// TIA Portal project "CAMASIR_MAKINASI" (V15.1)

(* hardware
DEVICE "S7300/ET200M station_1"  S7-300 station
   slot 0: "Rail_0"  Rail  6ES7 390-1***0-0AA0
   slot 2: "PLC_1"  CPU 314C-2 PN/DP  6ES7 314-6EH04-0AB0  V3.3
      slot 2: "PROFINET interface_1"  PN-IO
         slot 1: "Port_1"  Port
         slot 2: "Port_2"  Port
      slot 5: "DI 24/DO 16_1"  DI24/DO16
      slot 6: "AI 5/AO 2_1"  AI5/AO2
      slot 7: "Count_1"  Counter
      slot 8: "Positioning_1"  Positioning
*)

// ===== PLC "PLC_1"  CPU 314C-2 PN/DP =====

VAR_GLOBAL   // PLC tag table "Default tag table"
   "START" AT %I0.0 : Bool;
   "LAMBA" AT %Q0.0 : Bool;
   "STOP" AT %I0.1 : Bool;
   "V1" AT %Q0.1 : Bool;
   "L" AT %I0.2 : Bool;
   "H" AT %I0.3 : Bool;
   "Tag_1" AT %M0.0 : Bool;
   "Tag_2" AT %M1.0 : Bool;
   "Tag_3" AT %M0.1 : Bool;
   "Tag_4" AT %M1.1 : Bool;
   "Tag_5" AT %I0.7 : Bool;
   "Tag_6" AT %MW1 : Int;
   "V3" AT %Q0.2 : Bool;
   "L1" AT %I0.4 : Bool;
   "H1" AT %I0.5 : Bool;
   "Tag_7" AT %M0.2 : Bool;
   "Tag_8" AT %M1.2 : Bool;
   "Tag_9" AT %I0.6 : Bool;
   "Tag_10" AT %M0.3 : Bool;
   "Tag_11" AT %M1.3 : Bool;
   "M1" AT %Q0.3 : Bool;
   "L2" AT %I1.0 : Bool;
   "H2" AT %I1.1 : Bool;
   "Tag_12" AT %M0.4 : Bool;
   "Tag_13" AT %M1.4 : Bool;
   "Tag_14" AT %M0.5 : Bool;
   "Tag_15" AT %M1.5 : Bool;
   "V2" AT %Q0.6 : Bool;
   "L3" AT %I1.2 : Bool;
   "H3" AT %I1.3 : Bool;
   "Tag_16" AT %M0.6 : Bool;
   "Tag_17" AT %M1.6 : Bool;
   "Tag_18" AT %MW2 : Int;
   "Tag_19" AT %M2.2 : Bool;
   "Tag_20" AT %M2.3 : Bool;
   "Tag_21" AT %MW3 : Int;
   "Tag_22" AT %M1.7 : Bool;
   "Tag_23" AT %M2.0 : Bool;
   "Tag_24" AT %M2.1 : Bool;
END_VAR

ORGANIZATION_BLOCK "Main"   // OB1, LAD
TITLE = "Main Program Sweep (Cycle)"
{ S7_Optimized_Access := 'FALSE' }
VERSION : 0.1
   VAR_TEMP
      OB1_EV_CLASS : Byte;   // Bits 0-3 = 1 (Coming event), Bits 4-7 = 1 (Event class 1)
      OB1_SCAN_1 : Byte;   // 1 (Cold restart scan 1 of OB 1), 3 (Scan 2-n of OB 1)
      OB1_PRIORITY : Byte;   // Priority of OB Execution
      OB1_OB_NUMBR : Byte;   // 1 (Organization block 1, OB1)
      OB1_RESERVED_1 : Byte;   // Reserved for system
      OB1_RESERVED_2 : Byte;   // Reserved for system
      OB1_PREV_CYCLE : Int;   // Cycle time of previous OB1 scan (milliseconds)
      OB1_MIN_CYCLE : Int;   // Minimum cycle time of OB1 (milliseconds)
      OB1_MAX_CYCLE : Int;   // Maximum cycle time of OB1 (milliseconds)
      OB1_DATE_TIME : Date_And_Time;   // Date and time OB1 started
   END_VAR
   VAR_TEMP   // added for the SCL form of the ladder/FBD networks
      _w1 : Bool;
   END_VAR
BEGIN

REGION Network 1
   // START LAMA
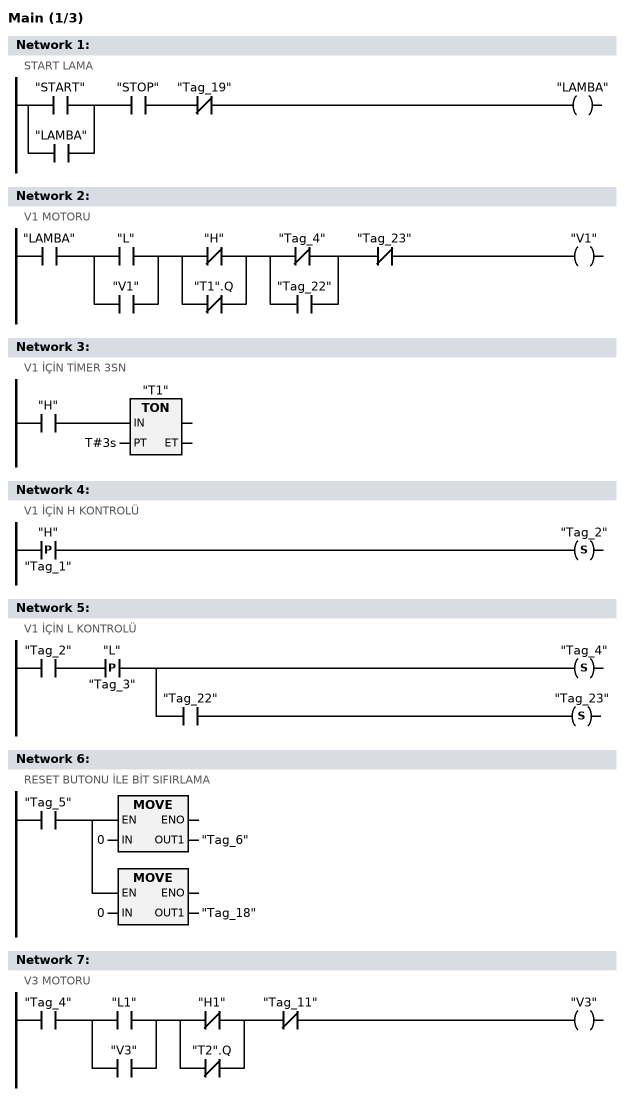
   RUNG wire#powerrail
      Contact( "START" )
      wire#w1
      Contact( "STOP" )
      I_Contact( "Tag_19" )
      Coil( "LAMBA" )
   END_RUNG
   RUNG wire#powerrail
      Contact( "LAMBA" )
   END_RUNG wire#w1
   // the same network as SCL:
   "LAMBA" := ("START" OR "LAMBA") AND "STOP" AND NOT "Tag_19";
END_REGION

REGION Network 2
   // V1 MOTORU
   RUNG wire#powerrail
      Contact( "LAMBA" )
      wire#w1
      Contact( "L" )
      wire#w2
      I_Contact( "H" )
      wire#w3
      I_Contact( "Tag_4" )
      wire#w4
      I_Contact( "Tag_23" )
      Coil( "V1" )
   END_RUNG
   RUNG wire#w1
      Contact( "V1" )
   END_RUNG wire#w2
   RUNG wire#w2
      I_Contact( "T1".Q )
   END_RUNG wire#w3
   RUNG wire#w3
      Contact( "Tag_22" )
   END_RUNG wire#w4
   // the same network as SCL:
   "V1" := "LAMBA" AND ("L" OR "V1") AND (NOT "H" OR NOT "T1".Q) AND (NOT "Tag_4" OR "Tag_22") AND NOT "Tag_23";
END_REGION

REGION Network 3
   // V1 İÇİN TİMER 3SN
   "T1".TON(IN := "H", PT := T#3s);
END_REGION

REGION Network 4
   // V1 İÇİN H KONTROLÜ
   RUNG wire#powerrail
      P_Contact(operand := "H", bit := "Tag_1")
      S_Coil( "Tag_2" )
   END_RUNG
   // the same network as SCL:
   #_w1 := "H" AND NOT "Tag_1";   // rising edge of "H"
   "Tag_1" := "H";
   IF #_w1 THEN "Tag_2" := TRUE; END_IF;
END_REGION

REGION Network 5
   // V1 İÇİN L KONTROLÜ
   RUNG wire#powerrail
      Contact( "Tag_2" )
      P_Contact(operand := "L", bit := "Tag_3")
      wire#w1
      S_Coil( "Tag_4" )
   END_RUNG
   RUNG wire#w1
      Contact( "Tag_22" )
      S_Coil( "Tag_23" )
   END_RUNG
   // the same network as SCL:
   #_w1 := "Tag_2" AND "L" AND NOT "Tag_3";   // rising edge of "L"
   "Tag_3" := "L";
   IF #_w1 THEN "Tag_4" := TRUE; END_IF;
   IF #_w1 AND "Tag_22" THEN "Tag_23" := TRUE; END_IF;
END_REGION

REGION Network 6
   // RESET BUTONU İLE BİT SIFIRLAMA
   RUNG wire#powerrail
      Contact( "Tag_5" )
      wire#w1
      { S7_GenerateENO := "TRUE" } Move(in := 0, out1 => "Tag_6")
   END_RUNG
   RUNG wire#w1
      { S7_GenerateENO := "TRUE" } Move(in := 0, out1 => "Tag_18")
   END_RUNG
   // the same network as SCL:
   IF "Tag_5" THEN
       "Tag_6" := 0;
       "Tag_18" := 0;
   END_IF;
END_REGION

REGION Network 7
   // V3 MOTORU
   RUNG wire#powerrail
      Contact( "Tag_4" )
      wire#w1
      Contact( "L1" )
      wire#w2
      I_Contact( "H1" )
      wire#w3
      I_Contact( "Tag_11" )
      Coil( "V3" )
   END_RUNG
   RUNG wire#w1
      Contact( "V3" )
   END_RUNG wire#w2
   RUNG wire#w2
      I_Contact( "T2".Q )
   END_RUNG wire#w3
   // the same network as SCL:
   "V3" := "Tag_4" AND ("L1" OR "V3") AND (NOT "H1" OR NOT "T2".Q) AND NOT "Tag_11";
END_REGION

REGION Network 8
   // V3 MOTORU İÇİN TİMER 5SN
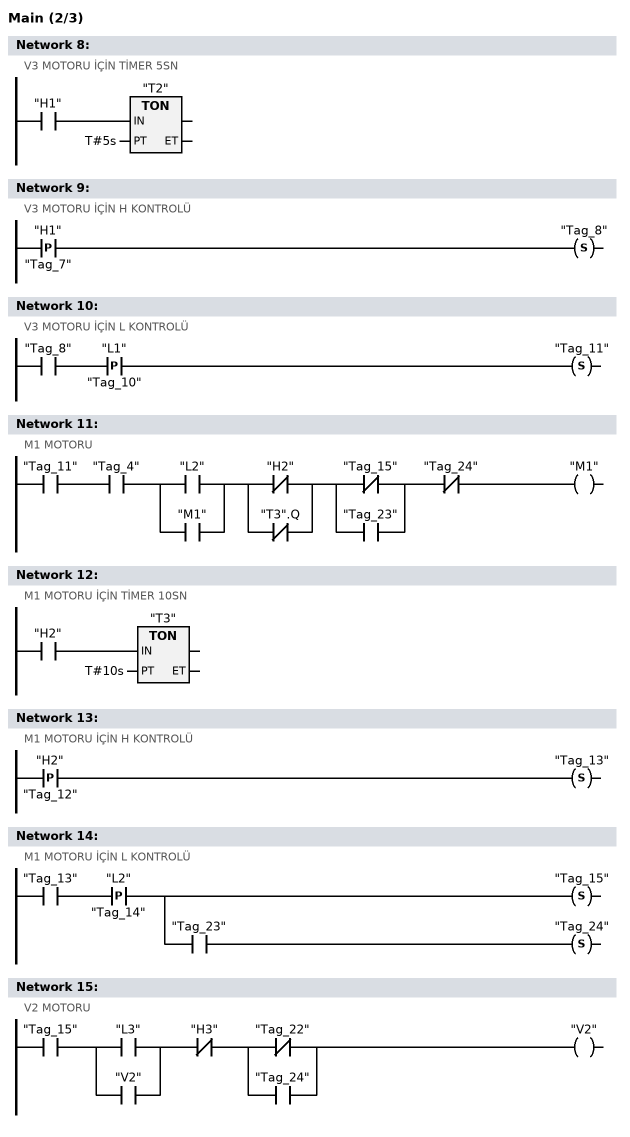
   "T2".TON(IN := "H1", PT := T#5s);
END_REGION

REGION Network 9
   // V3 MOTORU İÇİN H KONTROLÜ
   RUNG wire#powerrail
      P_Contact(operand := "H1", bit := "Tag_7")
      S_Coil( "Tag_8" )
   END_RUNG
   // the same network as SCL:
   #_w1 := "H1" AND NOT "Tag_7";   // rising edge of "H1"
   "Tag_7" := "H1";
   IF #_w1 THEN "Tag_8" := TRUE; END_IF;
END_REGION

REGION Network 10
   // V3 MOTORU İÇİN L KONTROLÜ
   RUNG wire#powerrail
      Contact( "Tag_8" )
      P_Contact(operand := "L1", bit := "Tag_10")
      S_Coil( "Tag_11" )
   END_RUNG
   // the same network as SCL:
   #_w1 := "Tag_8" AND "L1" AND NOT "Tag_10";   // rising edge of "L1"
   "Tag_10" := "L1";
   IF #_w1 THEN "Tag_11" := TRUE; END_IF;
END_REGION

REGION Network 11
   // M1 MOTORU
   RUNG wire#powerrail
      Contact( "Tag_11" )
      Contact( "Tag_4" )
      wire#w1
      Contact( "L2" )
      wire#w2
      I_Contact( "H2" )
      wire#w3
      I_Contact( "Tag_15" )
      wire#w4
      I_Contact( "Tag_24" )
      Coil( "M1" )
   END_RUNG
   RUNG wire#w1
      Contact( "M1" )
   END_RUNG wire#w2
   RUNG wire#w2
      I_Contact( "T3".Q )
   END_RUNG wire#w3
   RUNG wire#w3
      Contact( "Tag_23" )
   END_RUNG wire#w4
   // the same network as SCL:
   "M1" := "Tag_11" AND "Tag_4" AND ("L2" OR "M1") AND (NOT "H2" OR NOT "T3".Q) AND (NOT "Tag_15" OR "Tag_23") AND NOT "Tag_24";
END_REGION

REGION Network 12
   // M1 MOTORU İÇİN TİMER 10SN
   "T3".TON(IN := "H2", PT := T#10s);
END_REGION

REGION Network 13
   // M1 MOTORU İÇİN H KONTROLÜ
   RUNG wire#powerrail
      P_Contact(operand := "H2", bit := "Tag_12")
      S_Coil( "Tag_13" )
   END_RUNG
   // the same network as SCL:
   #_w1 := "H2" AND NOT "Tag_12";   // rising edge of "H2"
   "Tag_12" := "H2";
   IF #_w1 THEN "Tag_13" := TRUE; END_IF;
END_REGION

REGION Network 14
   // M1 MOTORU İÇİN L KONTROLÜ
   RUNG wire#powerrail
      Contact( "Tag_13" )
      P_Contact(operand := "L2", bit := "Tag_14")
      wire#w1
      S_Coil( "Tag_15" )
   END_RUNG
   RUNG wire#w1
      Contact( "Tag_23" )
      S_Coil( "Tag_24" )
   END_RUNG
   // the same network as SCL:
   #_w1 := "Tag_13" AND "L2" AND NOT "Tag_14";   // rising edge of "L2"
   "Tag_14" := "L2";
   IF #_w1 THEN "Tag_15" := TRUE; END_IF;
   IF #_w1 AND "Tag_23" THEN "Tag_24" := TRUE; END_IF;
END_REGION

REGION Network 15
   // V2 MOTORU
   RUNG wire#powerrail
      Contact( "Tag_15" )
      wire#w1
      Contact( "L3" )
      wire#w2
      I_Contact( "H3" )
      wire#w3
      I_Contact( "Tag_22" )
      wire#w4
      Coil( "V2" )
   END_RUNG
   RUNG wire#w1
      Contact( "V2" )
   END_RUNG wire#w2
   RUNG wire#w3
      Contact( "Tag_24" )
   END_RUNG wire#w4
   // the same network as SCL:
   "V2" := "Tag_15" AND ("L3" OR "V2") AND NOT "H3" AND (NOT "Tag_22" OR "Tag_24");
END_REGION

REGION Network 16
   // V2 MOTORU İÇİN H KONTOLÜ
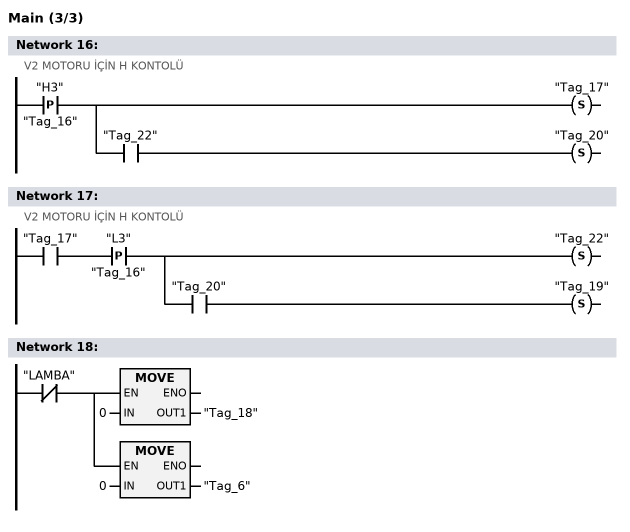
   RUNG wire#powerrail
      P_Contact(operand := "H3", bit := "Tag_16")
      wire#w1
      S_Coil( "Tag_17" )
   END_RUNG
   RUNG wire#w1
      Contact( "Tag_22" )
      S_Coil( "Tag_20" )
   END_RUNG
   // the same network as SCL:
   #_w1 := "H3" AND NOT "Tag_16";   // rising edge of "H3"
   "Tag_16" := "H3";
   IF #_w1 THEN "Tag_17" := TRUE; END_IF;
   IF #_w1 AND "Tag_22" THEN "Tag_20" := TRUE; END_IF;
END_REGION

REGION Network 17
   // V2 MOTORU İÇİN H KONTOLÜ
   RUNG wire#powerrail
      Contact( "Tag_17" )
      P_Contact(operand := "L3", bit := "Tag_16")
      wire#w1
      S_Coil( "Tag_22" )
   END_RUNG
   RUNG wire#w1
      Contact( "Tag_20" )
      S_Coil( "Tag_19" )
   END_RUNG
   // the same network as SCL:
   #_w1 := "Tag_17" AND "L3" AND NOT "Tag_16";   // rising edge of "L3"
   "Tag_16" := "L3";
   IF #_w1 THEN "Tag_22" := TRUE; END_IF;
   IF #_w1 AND "Tag_20" THEN "Tag_19" := TRUE; END_IF;
END_REGION

REGION Network 18
   RUNG wire#powerrail
      I_Contact( "LAMBA" )
      wire#w1
      { S7_GenerateENO := "TRUE" } Move(in := 0, out1 => "Tag_18")
   END_RUNG
   RUNG wire#w1
      { S7_GenerateENO := "TRUE" } Move(in := 0, out1 => "Tag_6")
   END_RUNG
   // the same network as SCL:
   IF NOT "LAMBA" THEN
       "Tag_18" := 0;
       "Tag_6" := 0;
   END_IF;
END_REGION
END_ORGANIZATION_BLOCK